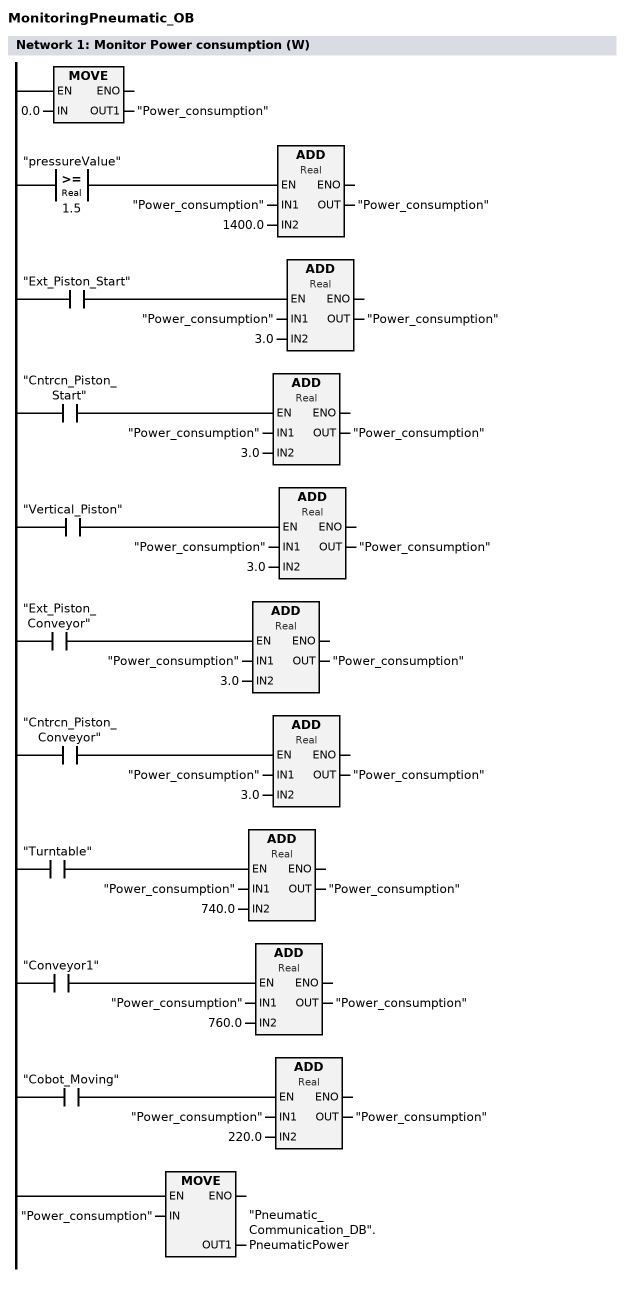
   RUNG wire#powerrail
      Move(in := 0.0, out1 => "Power_consumption")
   END_RUNG
   RUNG wire#powerrail
      { S7_Templates := "SrcType := Real" } GE_Contact(in1 := "pressureValue", in2 := 1.5)
      { S7_Templates := "SrcType := Real" } Add(in1 := "Power_consumption", in2 := 1400.0, out => "Power_consumption")
   END_RUNG
   RUNG wire#powerrail
      Contact( "Ext_Piston_Start" )
      { S7_Templates := "SrcType := Real" } Add(in1 := "Power_consumption", in2 := 3.0, out => "Power_consumption")
   END_RUNG
   RUNG wire#powerrail
      Contact( "Cntrcn_Piston_Start" )
      { S7_Templates := "SrcType := Real" } Add(in1 := "Power_consumption", in2 := 3.0, out => "Power_consumption")
   END_RUNG
   RUNG wire#powerrail
      Contact( "Vertical_Piston" )
      { S7_Templates := "SrcType := Real" } Add(in1 := "Power_consumption", in2 := 3.0, out => "Power_consumption")
   END_RUNG
   RUNG wire#powerrail
      Contact( "Ext_Piston_Conveyor" )
      { S7_Templates := "SrcType := Real" } Add(in1 := "Power_consumption", in2 := 3.0, out => "Power_consumption")
   END_RUNG
   RUNG wire#powerrail
      Contact( "Cntrcn_Piston_Conveyor" )
      { S7_Templates := "SrcType := Real" } Add(in1 := "Power_consumption", in2 := 3.0, out => "Power_consumption")
   END_RUNG
   RUNG wire#powerrail
      Contact( "Turntable" )
      { S7_Templates := "SrcType := Real" } Add(in1 := "Power_consumption", in2 := 740.0, out => "Power_consumption")
   END_RUNG
   RUNG wire#powerrail
      Contact( "Conveyor1" )
      { S7_Templates := "SrcType := Real" } Add(in1 := "Power_consumption", in2 := 760.0, out => "Power_consumption")
   END_RUNG
   RUNG wire#powerrail
      Contact( "Cobot_Moving" )
      { S7_Templates := "SrcType := Real" } Add(in1 := "Power_consumption", in2 := 220.0, out => "Power_consumption")
   END_RUNG
   RUNG wire#powerrail
      Move(in := "Power_consumption", out1 => "Pneumatic_Communication_DB".PneumaticPower)
   END_RUNG
   // the same network as SCL:
   "Power_consumption" := 0.0;
   IF "pressureValue" >= 1.5 THEN "Power_consumption" := "Power_consumption" + 1400.0; END_IF;
   IF "Ext_Piston_Start" THEN "Power_consumption" := "Power_consumption" + 3.0; END_IF;
   IF "Cntrcn_Piston_Start" THEN "Power_consumption" := "Power_consumption" + 3.0; END_IF;
   IF "Vertical_Piston" THEN "Power_consumption" := "Power_consumption" + 3.0; END_IF;
   IF "Ext_Piston_Conveyor" THEN "Power_consumption" := "Power_consumption" + 3.0; END_IF;
   IF "Cntrcn_Piston_Conveyor" THEN "Power_consumption" := "Power_consumption" + 3.0; END_IF;
   IF "Turntable" THEN "Power_consumption" := "Power_consumption" + 740.0; END_IF;
   IF "Conveyor1" THEN "Power_consumption" := "Power_consumption" + 760.0; END_IF;
   IF "Cobot_Moving" THEN "Power_consumption" := "Power_consumption" + 220.0; END_IF;
   "Pneumatic_Communication_DB".PneumaticPower := "Power_consumption";
END_REGION
END_ORGANIZATION_BLOCK

ORGANIZATION_BLOCK "RFID_OB"   // OB126, LAD, ProgramCycle
TITLE = "Main Program Sweep (Cycle)"
{ S7_Optimized_Access := 'TRUE' }
VERSION : 0.1
   VAR_INPUT
      Initial_Call : Bool;   // Initial call of this OB
      Remanence : Bool;   // =True, if remanent data are available
   END_VAR
   VAR_TEMP   // added for the SCL form of the ladder/FBD networks
      _w1 : Bool;
   END_VAR
BEGIN

REGION Network 1: Read nibble from RFID relay Device
   // K1 is LSB
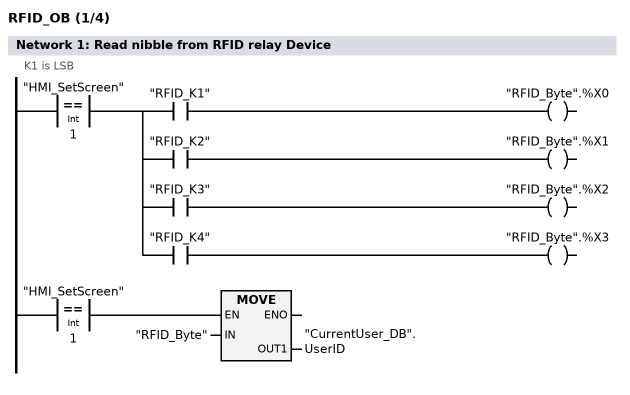
   RUNG wire#powerrail
      { S7_Templates := "SrcType := Int" } EQ_Contact(in1 := "HMI_SetScreen", in2 := 1)
      wire#w1
      Contact( "RFID_K1" )
      Coil( "RFID_Byte".%X0 )
   END_RUNG
   RUNG wire#w1
      Contact( "RFID_K2" )
      Coil( "RFID_Byte".%X1 )
   END_RUNG
   RUNG wire#w1
      Contact( "RFID_K3" )
      Coil( "RFID_Byte".%X2 )
   END_RUNG
   RUNG wire#w1
      Contact( "RFID_K4" )
      Coil( "RFID_Byte".%X3 )
   END_RUNG
   RUNG wire#powerrail
      { S7_Templates := "SrcType := Int" } EQ_Contact(in1 := "HMI_SetScreen", in2 := 1)
      Move(in := "RFID_Byte", out1 => "CurrentUser_DB".UserID)
   END_RUNG
   // the same network as SCL:
   #_w1 := "HMI_SetScreen" = 1;
   "RFID_Byte".%X0 := #_w1 AND "RFID_K1";
   "RFID_Byte".%X1 := #_w1 AND "RFID_K2";
   "RFID_Byte".%X2 := #_w1 AND "RFID_K3";
   "RFID_Byte".%X3 := #_w1 AND "RFID_K4";
   IF "HMI_SetScreen" = 1 THEN "CurrentUser_DB".UserID := "RFID_Byte"; END_IF;
END_REGION

REGION Network 2: Grant access and credentials
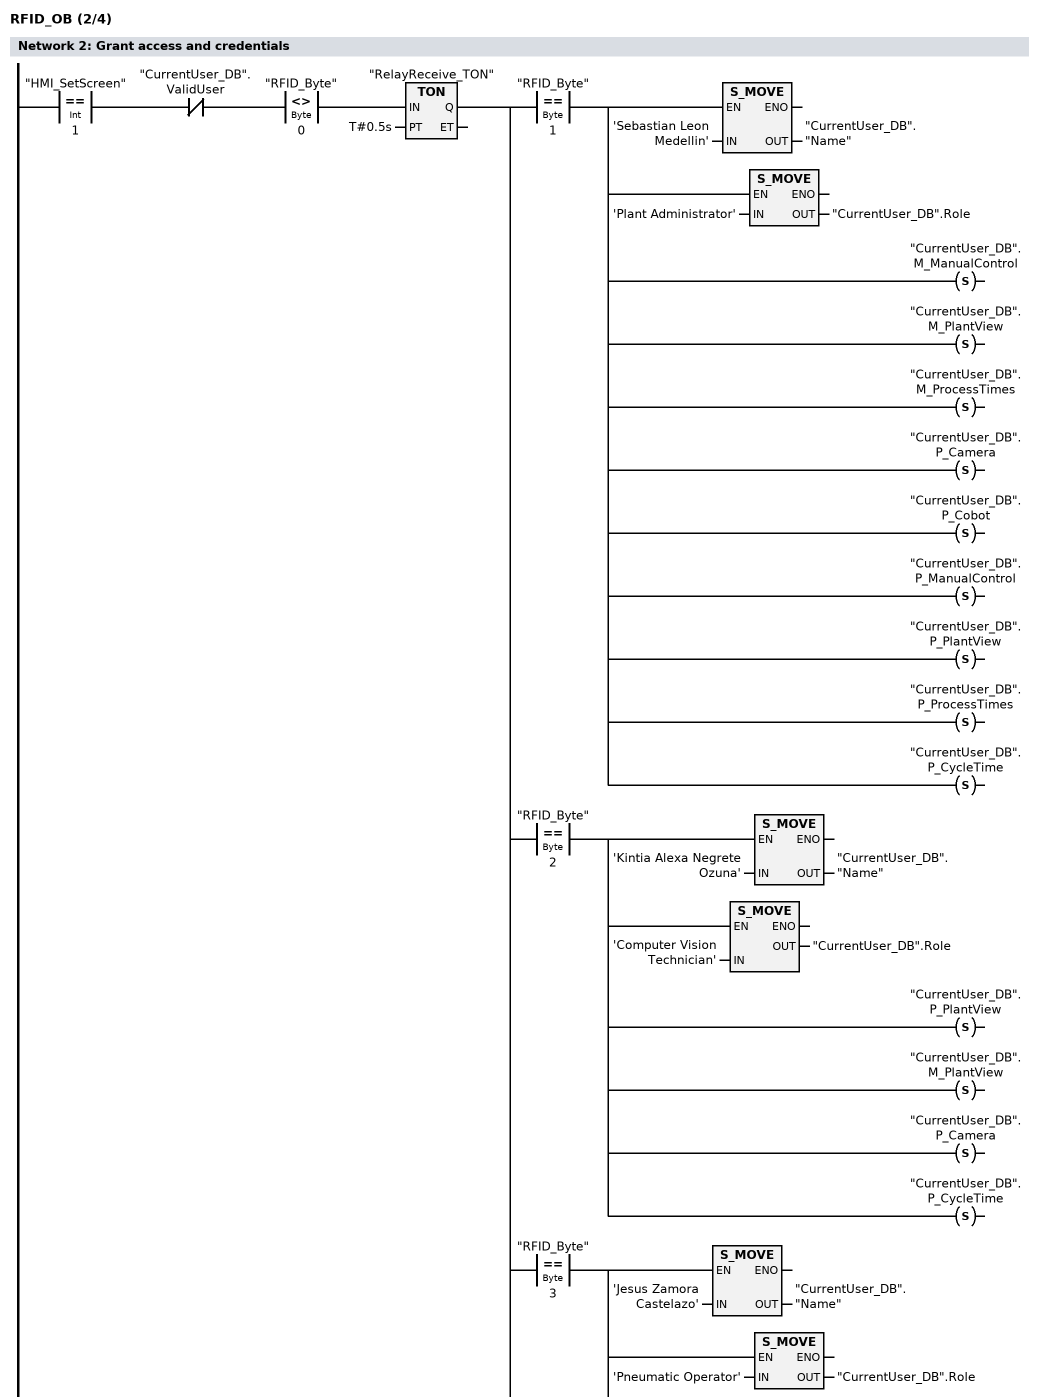
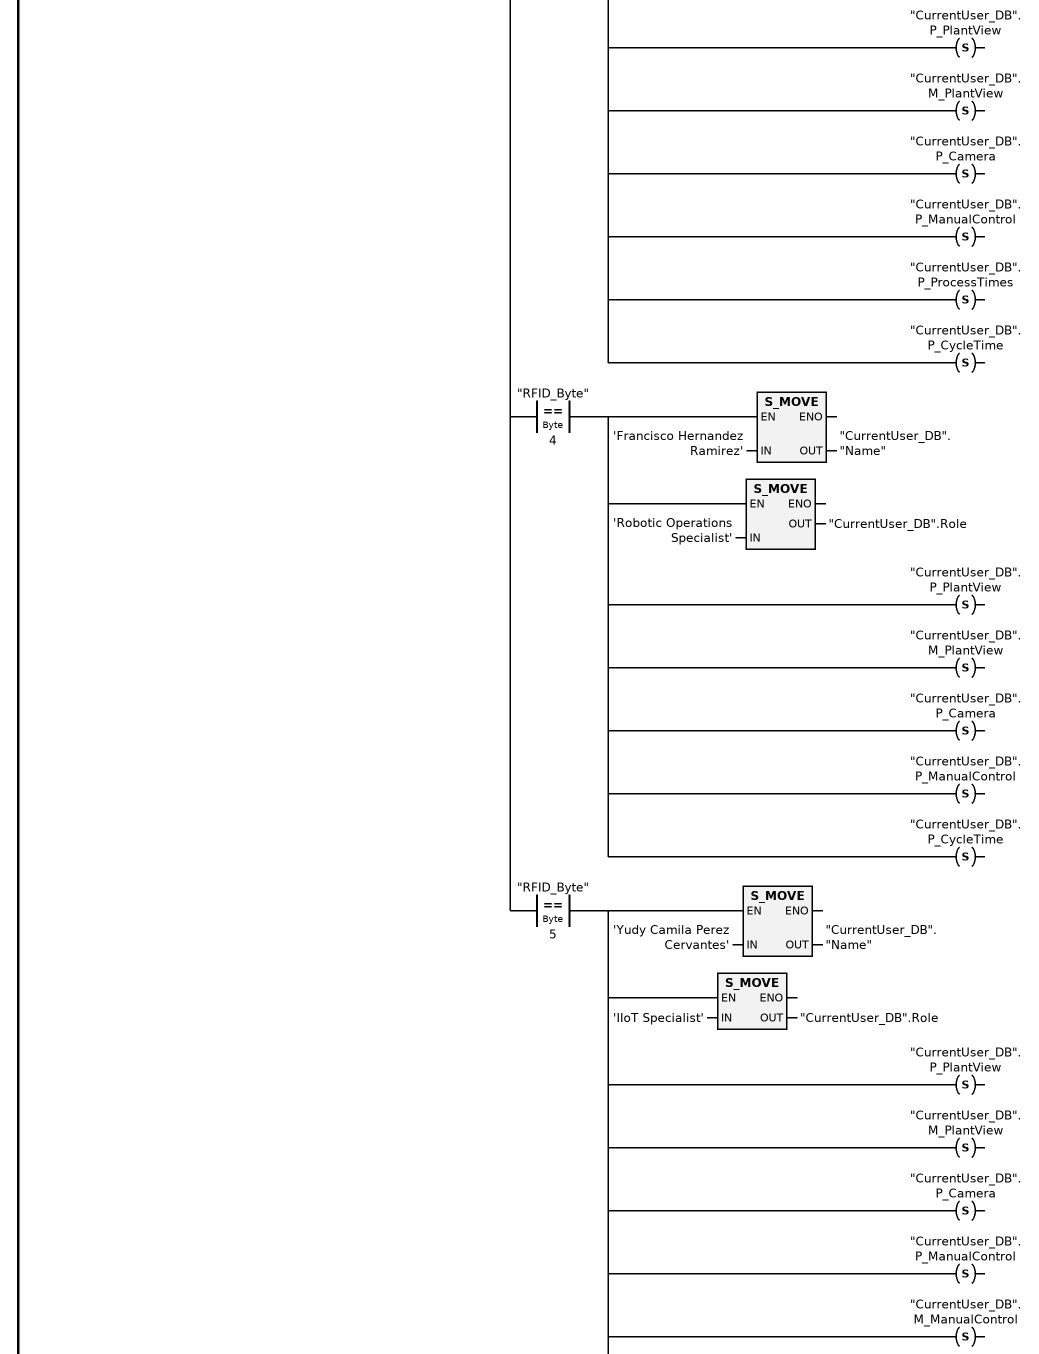
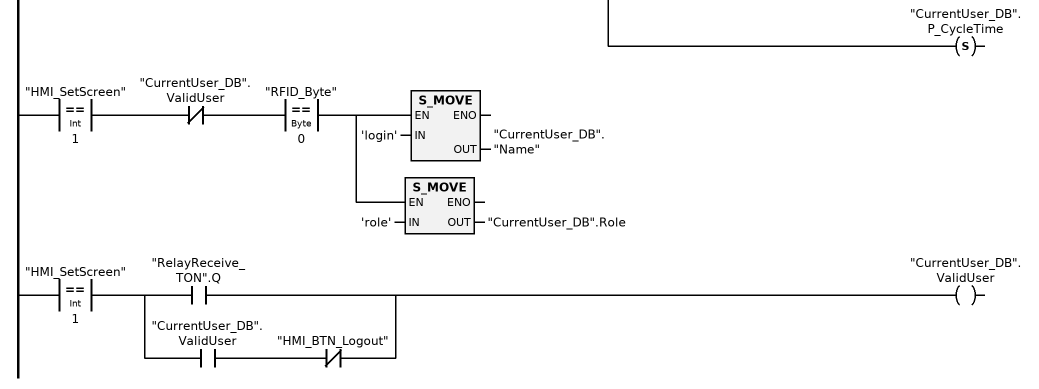
   "RelayReceive_TON".TON(IN := ("HMI_SetScreen" = 1) AND NOT "CurrentUser_DB".ValidUser AND ("RFID_Byte" <> 0),
                          PT := T#0.5s);
   IF "RelayReceive_TON".Q AND ("RFID_Byte" = 1) THEN
       "CurrentUser_DB"."Name" := 'Sebastian Leon Medellin';
       "CurrentUser_DB".Role := 'Plant Administrator';
       "CurrentUser_DB".M_ManualControl := TRUE;
       "CurrentUser_DB".M_PlantView := TRUE;
       "CurrentUser_DB".M_ProcessTimes := TRUE;
       "CurrentUser_DB".P_Camera := TRUE;
       "CurrentUser_DB".P_Cobot := TRUE;
       "CurrentUser_DB".P_ManualControl := TRUE;
       "CurrentUser_DB".P_PlantView := TRUE;
       "CurrentUser_DB".P_ProcessTimes := TRUE;
       "CurrentUser_DB".P_CycleTime := TRUE;
   END_IF;
   IF "RelayReceive_TON".Q AND ("RFID_Byte" = 2) THEN
       "CurrentUser_DB"."Name" := 'Kintia Alexa Negrete Ozuna';
       "CurrentUser_DB".Role := 'Computer Vision Technician';
       "CurrentUser_DB".P_PlantView := TRUE;
       "CurrentUser_DB".M_PlantView := TRUE;
       "CurrentUser_DB".P_Camera := TRUE;
       "CurrentUser_DB".P_CycleTime := TRUE;
   END_IF;
   IF "RelayReceive_TON".Q AND ("RFID_Byte" = 3) THEN
       "CurrentUser_DB"."Name" := 'Jesus Zamora Castelazo';
       "CurrentUser_DB".Role := 'Pneumatic Operator';
       "CurrentUser_DB".P_PlantView := TRUE;
       "CurrentUser_DB".M_PlantView := TRUE;
       "CurrentUser_DB".P_Camera := TRUE;
       "CurrentUser_DB".P_ManualControl := TRUE;
       "CurrentUser_DB".P_ProcessTimes := TRUE;
       "CurrentUser_DB".P_CycleTime := TRUE;
   END_IF;
   IF "RelayReceive_TON".Q AND ("RFID_Byte" = 4) THEN
       "CurrentUser_DB"."Name" := 'Francisco Hernandez Ramirez';
       "CurrentUser_DB".Role := 'Robotic Operations Specialist';
       "CurrentUser_DB".P_PlantView := TRUE;
       "CurrentUser_DB".M_PlantView := TRUE;
       "CurrentUser_DB".P_Camera := TRUE;
       "CurrentUser_DB".P_ManualControl := TRUE;
       "CurrentUser_DB".P_CycleTime := TRUE;
   END_IF;
   IF "RelayReceive_TON".Q AND ("RFID_Byte" = 5) THEN
       "CurrentUser_DB"."Name" := 'Yudy Camila Perez Cervantes';
       "CurrentUser_DB".Role := 'IIoT Specialist';
       "CurrentUser_DB".P_PlantView := TRUE;
       "CurrentUser_DB".M_PlantView := TRUE;
       "CurrentUser_DB".P_Camera := TRUE;
       "CurrentUser_DB".P_ManualControl := TRUE;
       "CurrentUser_DB".M_ManualControl := TRUE;
       "CurrentUser_DB".P_CycleTime := TRUE;
   END_IF;
   IF ("HMI_SetScreen" = 1) AND NOT "CurrentUser_DB".ValidUser AND ("RFID_Byte" = 0) THEN
       "CurrentUser_DB"."Name" := 'login';
       "CurrentUser_DB".Role := 'role';
   END_IF;
   "CurrentUser_DB".ValidUser := ("HMI_SetScreen" = 1) AND ("RelayReceive_TON".Q OR ("CurrentUser_DB".ValidUser AND NOT "HMI_BTN_Logout"));
END_REGION

REGION Network 3: Send user and role data trough S7
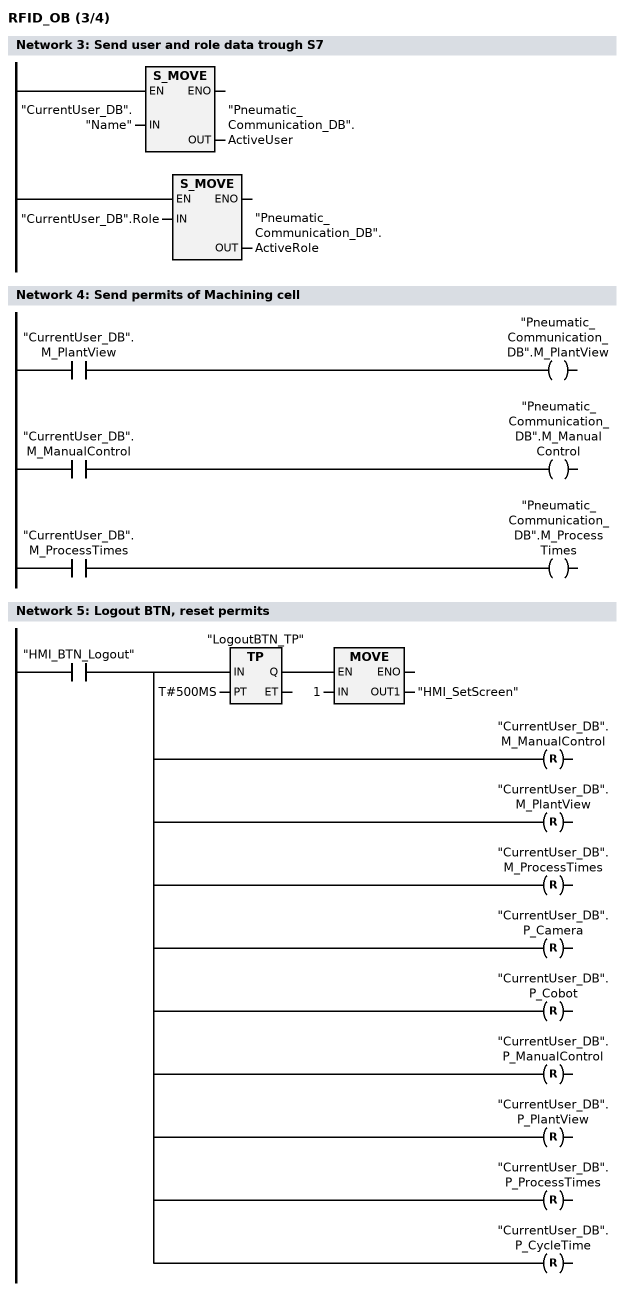
   RUNG wire#powerrail
      S_Move(in := "CurrentUser_DB"."Name", out => "Pneumatic_Communication_DB".ActiveUser)
   END_RUNG
   RUNG wire#powerrail
      S_Move(in := "CurrentUser_DB".Role, out => "Pneumatic_Communication_DB".ActiveRole)
   END_RUNG
   // the same network as SCL:
   "Pneumatic_Communication_DB".ActiveUser := "CurrentUser_DB"."Name";
   "Pneumatic_Communication_DB".ActiveRole := "CurrentUser_DB".Role;
END_REGION

REGION Network 4: Send permits of Machining cell
   RUNG wire#powerrail
      Contact( "CurrentUser_DB".M_PlantView )
      Coil( "Pneumatic_Communication_DB".M_PlantView )
   END_RUNG
   RUNG wire#powerrail
      Contact( "CurrentUser_DB".M_ManualControl )
      Coil( "Pneumatic_Communication_DB".M_ManualControl )
   END_RUNG
   RUNG wire#powerrail
      Contact( "CurrentUser_DB".M_ProcessTimes )
      Coil( "Pneumatic_Communication_DB".M_ProcessTimes )
   END_RUNG
   // the same network as SCL:
   "Pneumatic_Communication_DB".M_PlantView := "CurrentUser_DB".M_PlantView;
   "Pneumatic_Communication_DB".M_ManualControl := "CurrentUser_DB".M_ManualControl;
   "Pneumatic_Communication_DB".M_ProcessTimes := "CurrentUser_DB".M_ProcessTimes;
END_REGION

REGION Network 5: Logout BTN, reset permits
   "LogoutBTN_TP".TP(IN := "HMI_BTN_Logout", PT := T#500MS);
   IF "LogoutBTN_TP".Q THEN "HMI_SetScreen" := 1; END_IF;
   IF "HMI_BTN_Logout" THEN
       "CurrentUser_DB".M_ManualControl := FALSE;
       "CurrentUser_DB".M_PlantView := FALSE;
       "CurrentUser_DB".M_ProcessTimes := FALSE;
       "CurrentUser_DB".P_Camera := FALSE;
       "CurrentUser_DB".P_Cobot := FALSE;
       "CurrentUser_DB".P_ManualControl := FALSE;
       "CurrentUser_DB".P_PlantView := FALSE;
       "CurrentUser_DB".P_ProcessTimes := FALSE;
       "CurrentUser_DB".P_CycleTime := FALSE;
   END_IF;
END_REGION

REGION Network 6: Send logout bit
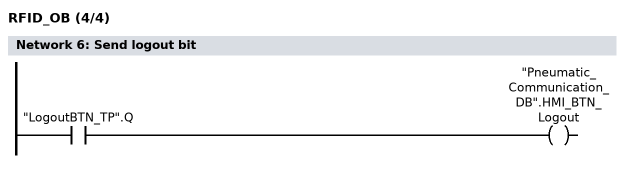
   RUNG wire#powerrail
      Contact( "LogoutBTN_TP".Q )
      Coil( "Pneumatic_Communication_DB".HMI_BTN_Logout )
   END_RUNG
   // the same network as SCL:
   "Pneumatic_Communication_DB".HMI_BTN_Logout := "LogoutBTN_TP".Q;
END_REGION
END_ORGANIZATION_BLOCK

ORGANIZATION_BLOCK "CycleTime_OB"   // OB127, LAD, ProgramCycle
TITLE = "Main Program Sweep (Cycle)"
{ S7_Optimized_Access := 'TRUE' }
VERSION : 0.1
   VAR_INPUT
      Initial_Call : Bool;   // Initial call of this OB
      Remanence : Bool;   // =True, if remanent data are available
   END_VAR
BEGIN

REGION Network 1: Enabled Measuring latch
   // This latch confirms that the PLC is either
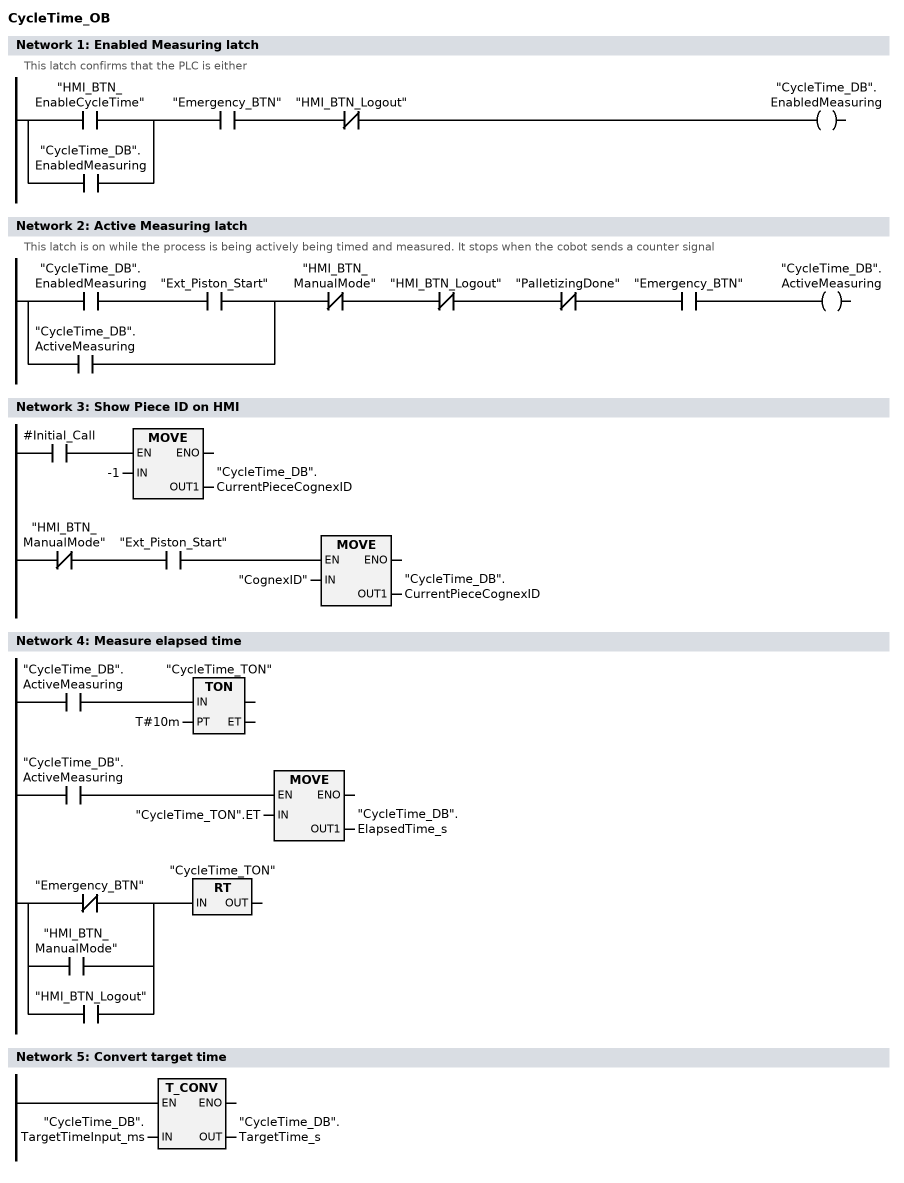
   RUNG wire#powerrail
      Contact( "HMI_BTN_EnableCycleTime" )
      wire#w1
      Contact( "Emergency_BTN" )
      I_Contact( "HMI_BTN_Logout" )
      Coil( "CycleTime_DB".EnabledMeasuring )
   END_RUNG
   RUNG wire#powerrail
      Contact( "CycleTime_DB".EnabledMeasuring )
   END_RUNG wire#w1
   // the same network as SCL:
   "CycleTime_DB".EnabledMeasuring := ("HMI_BTN_EnableCycleTime" OR "CycleTime_DB".EnabledMeasuring) AND "Emergency_BTN" AND NOT "HMI_BTN_Logout";
END_REGION

REGION Network 2: Active Measuring latch
   // This latch is on while the process is being actively being timed and measured. It stops when the cobot sends a counter signal
   RUNG wire#powerrail
      Contact( "CycleTime_DB".EnabledMeasuring )
      Contact( "Ext_Piston_Start" )
      wire#w1
      I_Contact( "HMI_BTN_ManualMode" )
      I_Contact( "HMI_BTN_Logout" )
      I_Contact( "PalletizingDone" )
      Contact( "Emergency_BTN" )
      Coil( "CycleTime_DB".ActiveMeasuring )
   END_RUNG
   RUNG wire#powerrail
      Contact( "CycleTime_DB".ActiveMeasuring )
   END_RUNG wire#w1
   // the same network as SCL:
   "CycleTime_DB".ActiveMeasuring := (("CycleTime_DB".EnabledMeasuring AND "Ext_Piston_Start") OR "CycleTime_DB".ActiveMeasuring) AND NOT "HMI_BTN_ManualMode" AND NOT "HMI_BTN_Logout" AND NOT "PalletizingDone" AND "Emergency_BTN";
END_REGION

REGION Network 3: Show Piece ID on HMI
   RUNG wire#powerrail
      Contact( #Initial_Call )
      Move(in := -1, out1 => "CycleTime_DB".CurrentPieceCognexID)
   END_RUNG
   RUNG wire#powerrail
      I_Contact( "HMI_BTN_ManualMode" )
      Contact( "Ext_Piston_Start" )
      Move(in := "CognexID", out1 => "CycleTime_DB".CurrentPieceCognexID)
   END_RUNG
   // the same network as SCL:
   IF #Initial_Call THEN "CycleTime_DB".CurrentPieceCognexID := -1; END_IF;
   IF NOT "HMI_BTN_ManualMode" AND "Ext_Piston_Start" THEN
       "CycleTime_DB".CurrentPieceCognexID := "CognexID";
   END_IF;
END_REGION

REGION Network 4: Measure elapsed time
   "CycleTime_TON".TON(IN := "CycleTime_DB".ActiveMeasuring, PT := T#10m);
   IF "CycleTime_DB".ActiveMeasuring THEN "CycleTime_DB".ElapsedTime_s := "CycleTime_TON".ET; END_IF;
   IF NOT "Emergency_BTN" OR "HMI_BTN_ManualMode" OR "HMI_BTN_Logout" THEN
       RESET_TIMER("CycleTime_TON");
   END_IF;
END_REGION

REGION Network 5: Convert target time
   "CycleTime_DB".TargetTime_s := T_CONV(IN := "CycleTime_DB".TargetTimeInput_ms);
END_REGION
END_ORGANIZATION_BLOCK

(* ===== HMI "HMI_RT_1" =====
system functions are stored by id; their names below are inferred from use
connection "HMI_Connection_1": ETHERNET, SMART_S7_1200_OMS

HMI tags "Default tag table"
   "Tag_ScreenNumber" : UInt, internal
   "HMI_BTN1" : Bool = PLC HMI_BTN1 AT %M50.0, 100 ms
   "Conveyor2" : Bool = PLC Conveyor2 AT %Q0.0, 100 ms
   "Pusher1" : Bool = PLC Pusher1 AT %Q0.1, 100 ms
   "Drill" : Bool = PLC Drill AT %Q0.3, 100 ms
   "Mix" : Bool = PLC Mix AT %Q0.5, 100 ms
   "Pusher2" : Bool = PLC Pusher2 AT %Q0.6, 500 ms
   "Conveyor5" : Bool = PLC Conveyor5 AT %Q0.7, 100 ms
   "Conveyor6_OUT" : Bool = PLC Conveyor6_OUT AT %Q8.3, 100 ms
   "Conveyor6_IN" : Bool = PLC Conveyor6_IN AT %Q8.2, 100 ms
   "Red_Tower" : Bool = PLC Red_Tower AT %Q1.1, 500 ms
   "Green_Tower" : Bool = PLC Green_Tower AT %Q1.0, 100 ms
   "cakeFlavor" : UInt = PLC cakeFlavor AT %MW12, 100 ms
   "Conveyor3" : Bool = PLC Conveyor3 AT %Q0.2, 100 ms
   "Conveyor4" : Bool = PLC Conveyor4 AT %Q0.4, 100 ms
   "Press_UP" : Bool = PLC Press_UP AT %Q8.4, 100 ms
   "Press_DOWN" : Bool = PLC Press_DOWN AT %Q8.5, 100 ms
   "drillingTime" : Time = PLC drillingTime AT %MD14, 100 ms
   "processTimes_DB_chocolateDrillingInput" : UInt = PLC processTimes_DB.chocolateDrillingInput_ms, 1 s
   "processTimes_DB_chocolateMixingInput" : UInt = PLC processTimes_DB.chocolateMixingInput_ms, 1 s
   "processTimes_DB_vanillaDrillingInput_ms" : UInt = PLC processTimes_DB.vanillaDrillingInput_ms, 1 s
   "processTimes_DB_vamillaMixingInput_ms" : UInt = PLC processTimes_DB.vanillaMixingInput_ms, 1 s
   "processTimes_DB_strawberryDrillingInput_ms" : UInt = PLC processTimes_DB.strawberryDrillingInput_ms, 1 s
   "processTimes_DB_strawberryMixingInput_ms" : UInt = PLC processTimes_DB.strawberryMixingInput_ms, 1 s
   "ManualMode_SW" : Bool = PLC ManualMode_SW AT %M53.0, 100 ms
   "HMI_BTN_Conveyor2" : Bool = PLC HMI_BTN_Conveyor2 AT %M50.1, 100 ms
   "HMI_BTN_Pusher1" : Bool = PLC HMI_BTN_Pusher1 AT %M50.2, 100 ms
   "HMI_BTN_Conveyor3" : Bool = PLC HMI_BTN_Conveyor3 AT %M50.3, 100 ms
   "HMI_BTN_Conveyor4" : Bool = PLC HMI_BTN_Conveyor4 AT %M50.4, 100 ms
   "HMI_BTN_Drill" : Bool = PLC HMI_BTN_Drill AT %M50.6, 100 ms
   "HMI_BTN_Mix" : Bool = PLC HMI_BTN_Mix AT %M50.7, 100 ms
   "HMI_BTN_Conveyor5" : Bool = PLC HMI_BTN_Conveyor5 AT %M50.5, 100 ms
   "HMI_BTN_Pusher2" : Bool = PLC HMI_BTN_Pusher2 AT %M51.0, 100 ms
   "HMI_BTN_Conveyor6IN" : Bool = PLC HMI_BTN_Conveyor6IN AT %M51.1, 100 ms
   "HMI_BTN_Conveyor6OUT" : Bool = PLC HMI_BTN_Conveyor6OUT AT %M51.2, 100 ms
   "HMI_BTN_PressDown" : Bool = PLC HMI_BTN_PressDown AT %M51.3, 100 ms
   "HMI_BTN_PressUp" : Bool = PLC HMI_BTN_PressUp AT %M51.4, 100 ms
   "Power_consumption" : Real = PLC Power_consumption AT %MD28, 100 ms
   "HMI_SetScreen" : Int = PLC HMI_SetScreen AT %MW54, 100 ms
      on ChangeValue: ActivateScreenByNumber("HMI_SetScreen", 0)
   "HMI_BTN_PlantView" : Bool = PLC HMI_BTN_PlantView AT %M51.5, 100 ms
   "HMI_BTN_ProcessTimes" : Bool = PLC HMI_BTN_ProcessTimes AT %M51.6, 100 ms
   "HMI_BTN_ManualControl" : Bool = PLC HMI_BTN_ManualControl AT %M51.7, 100 ms
   "Machining_Communication_DB_M_PlantView" : Bool = PLC Machining_Communication_DB.M_PlantView AT %DB100.DBX5.5, 1 s
   "Machining_Communication_DB_M_ProcessTimes" : Bool = PLC Machining_Communication_DB.M_ProcessTimes AT %DB100.DBX5.7, 1 s
   "Machining_Communication_DB_M_ManualControl" : Bool = PLC Machining_Communication_DB.M_ManualControl AT %DB100.DBX5.6, 1 s

text list "Flavors": 0 'Chocolate'; 1 'Vanilla'; 2 'Strawberry'; 4 'Flavor'; -1 'NA'

Template "Template_1" 800x480
   TextField "Template_Text field_1" at 62,8 size 412x56; Text 'MR2007B Automation of Manufacturing Systems ATOLE S.A. de C.V.'
   GraphicView "Template_Graphic view_1" at 529,9 size 252x54; Picture "eic"
   GraphicView "Template_Graphic view_2" at 21,13 size 34x45; Picture "atoleLogo_transparent"

screen "Root screen" 800x480, template "Template_1"
   TextField "HmiScreenItemData" at 40,88 size 720x57; Text 'Welcome to ATOLE S.A. de C.V.'
   Button "Button_2" at 136,208 size 240x56; TextOff 'Plant View'
      on Press: SetBit("HMI_BTN_PlantView")
      on Release: ResetBit("HMI_BTN_PlantView")
   GraphicView "Graphic view_1" at 429,152 size 294x294; Picture "cake"
   Button "Button_3" at 136,280 size 240x56; TextOff 'Set Process Times'
      on Press: SetBit("HMI_BTN_ProcessTimes")
      on Release: ResetBit("HMI_BTN_ProcessTimes")
   Button "Button_4" at 136,352 size 240x56; TextOff 'Manual Control'
      on Press: SetBit("HMI_BTN_ManualControl")
      on Release: ResetBit("HMI_BTN_ManualControl")
   Rectangle "Rectangle_1" at 144,216 size 40x40
      Appearance <- "Machining_Communication_DB_M_PlantView"
   Rectangle "Rectangle_2" at 144,288 size 40x40
      Appearance <- "Machining_Communication_DB_M_ProcessTimes"
   Rectangle "Rectangle_3" at 144,360 size 40x40
      Appearance <- "Machining_Communication_DB_M_ManualControl"

screen "PlantView" 800x480, template "Template_1"
   GraphicView "Graphic view_1" at 14,74 size 773x401; Picture "machiningCellDiagram_2"
   Circle "Circle_1" at 684,86 size 11x11
      Visibility <- "Conveyor2"
   Circle "Circle_2" at 747,252 size 11x11
      Visibility <- "Pusher1"
   Circle "Circle_3" at 546,386 size 11x11
      Visibility <- "Drill"
   Circle "Circle_4" at 323,435 size 11x11
      Visibility <- "Pusher2"
   Circle "Circle_5" at 342,144 size 11x11
      Visibility <- "Conveyor5"
   Circle "Circle_6" at 400,386 size 11x11
      Visibility <- "Mix"
   GraphicView "Graphic view_2" at 33,112 size 21x24; Picture "arrow"
      Visibility <- "Conveyor6_OUT"
   GraphicView "Graphic view_3" at 33,186 size 21x24; Picture "arrowDown"
      Visibility <- "Conveyor6_IN"
   Rectangle "Rectangle_1" at 670,360 size 20x20
      Visibility <- "Red_Tower"
   Rectangle "Rectangle_2" at 699,360 size 20x20
      Visibility <- "Green_Tower"
   TextField "Text field_1" at 319,72 size 162x39; Text 'Plant View'
   Circle "Circle_7" at 556,194 size 11x11
      Visibility <- "Conveyor3"
   Circle "Circle_8" at 417,194 size 11x11
      Visibility <- "Conveyor4"
   GraphicView "Graphic view_4" at 33,361 size 21x24; Picture "arrowDown"
      Visibility <- "Press_DOWN"
   GraphicView "Graphic view_5" at 33,286 size 21x24; Picture "arrow"
      Visibility <- "Press_UP"
   IOField "I/O field_1" at 600,432 size 184x32; FormatPattern 999999999999; Unit  W
      ProcessValue <- "Power_consumption"
   TextField "Text field_2" at 616,408 size 168x23; Text 'Power Consumption'
   Button "Button_1" at 16,424 size 104x40; TextOff 'Home'
      on Press: ActivateScreen("Root screen", 0); SetTag("HMI_SetScreen", 2)

screen "ManualControl" 800x480, template "Template_1"
   Switch "Switch_1" at 84,224 size 120x56; CaptionText 'Switch'; TextOff 'OFF'; TextOn 'ON'
      ProcessValue <- "ManualMode_SW"
      on SwitchOn: SetBit("ManualMode_SW")
      on SwitchOff: ResetBit("ManualMode_SW")
   TextField "Text field_2" at 84,284 size 121x36; Text 'Enable manual control'
   Button "Button_2" at 252,144 size 144x32; TextOff 'Conveyor 2'
      on Press: SetBit("HMI_BTN_Conveyor2")
      on Release: ResetBit("HMI_BTN_Conveyor2")
   Button "Button_3" at 252,192 size 144x32; TextOff 'Pusher 1'
      on Press: SetBit("HMI_BTN_Pusher1")
      on Release: ResetBit("HMI_BTN_Pusher1")
   Button "Button_4" at 252,240 size 144x32; TextOff 'Conveyor 3'
      on Release: ResetBit("HMI_BTN_Conveyor3")
      on Press: SetBit("HMI_BTN_Conveyor3")
   Button "Button_5" at 252,288 size 144x32; TextOff 'Conveyor 4'
      on Press: SetBit("HMI_BTN_Conveyor4")
      on Release: ResetBit("HMI_BTN_Conveyor4")
   Button "Button_6" at 252,336 size 144x32; TextOff 'Drill'
      on Press: SetBit("HMI_BTN_Drill")
      on Release: ResetBit("HMI_BTN_Drill")
   Button "Button_7" at 252,384 size 144x32; TextOff 'Mix'
      on Press: SetBit("HMI_BTN_Mix")
      on Release: ResetBit("HMI_BTN_Mix")
   Button "Button_8" at 524,144 size 144x32; TextOff 'Pusher 2'
      on Press: SetBit("HMI_BTN_Pusher2")
      on Release: ResetBit("HMI_BTN_Pusher2")
   Button "Button_9" at 524,192 size 144x32; TextOff 'Conveyor 5'
      on Press: SetBit("HMI_BTN_Conveyor5")
      on Release: ResetBit("HMI_BTN_Conveyor5")
   Circle "Circle_1" at 412,144 size 32x32
      Appearance <- "Conveyor2"
   Circle "Circle_2" at 412,192 size 32x32
      Appearance <- "Pusher1"
   Circle "Circle_3" at 412,240 size 32x32
      Appearance <- "Conveyor3"
   Circle "Circle_4" at 412,288 size 32x32
      Appearance <- "Conveyor4"
   Circle "Circle_5" at 412,336 size 32x32
      Appearance <- "Drill"
   Circle "Circle_6" at 412,384 size 32x32
      Appearance <- "Mix"
   Circle "Circle_7" at 684,144 size 32x32
      Appearance <- "Pusher2"
   Circle "Circle_8" at 684,192 size 32x32
      Appearance <- "Conveyor5"
   Button "Button_10" at 524,240 size 144x32; TextOff 'Conveyor 6 IN'
      on Press: SetBit("HMI_BTN_Conveyor6IN")
      on Release: ResetBit("HMI_BTN_Conveyor6IN")
   Button "Button_11" at 524,288 size 144x32; TextOff 'Conveyor 6 OUT'
      on Press: SetBit("HMI_BTN_Conveyor6OUT")
      on Release: ResetBit("HMI_BTN_Conveyor6OUT")
   Button "Button_12" at 524,336 size 144x32; TextOff 'Press Down'
      on Press: SetBit("HMI_BTN_PressDown")
      on Release: ResetBit("HMI_BTN_PressDown")
   Button "Button_13" at 524,384 size 144x32; TextOff 'Press Up'
      on Press: SetBit("HMI_BTN_PressUp")
      on Release: ResetBit("HMI_BTN_PressUp")
   Circle "Circle_9" at 684,240 size 32x32
      Appearance <- "Conveyor6_IN"
   Circle "Circle_10" at 684,288 size 32x32
      Appearance <- "Conveyor6_OUT"
   Circle "Circle_11" at 684,336 size 32x32
      Appearance <- "Press_DOWN"
   Circle "Circle_12" at 684,384 size 32x32
      Appearance <- "Press_UP"
   Button "Button_1" at 16,424 size 104x40; TextOff 'Home'
      on Press: ActivateScreen("Root screen", 0); SetTag("HMI_SetScreen", 2)
   TextField "Text field_1" at 208,80 size 389x39; Text 'Machining Manual Control'
   Group "Group" at 84,144 size 632x272
   TextField "Text field_4" at 400,432 size 393x48; Text 'Manual Mode: Press and hold the button to actuate'

screen "ProcessTimes" 800x480, template "Template_1"
   TextField "Text field_1" at 294,88 size 213x39; Text 'Process Times'
   Button "Button_1" at 16,424 size 104x40; TextOff 'Home'
      on Press: ActivateScreen("Root screen", 0); SetTag("HMI_SetScreen", 2)
   TextField "Text field_5" at 74,208 size 104x48; Text 'Drilling'
   TextField "Text field_6" at 82,280 size 96x48; Text 'Mixing'
   IOField "I/O field_1" at 190,208 size 152x48; FormatPattern 9999999; Unit  s
      ProcessValue <- "processTimes_DB_chocolateDrillingInput"
   IOField "I/O field_2" at 190,280 size 152x48; FormatPattern 9999999; Unit  s
      ProcessValue <- "processTimes_DB_chocolateMixingInput"
   TextField "Text field_2" at 190,168 size 156x34; Text 'Chocolate'
   TextField "Text field_3" at 382,168 size 156x34; Text 'Vanilla'
   TextField "Text field_4" at 574,168 size 152x31; Text 'Strawberry'
   IOField "I/O field_3" at 382,280 size 152x48; FormatPattern 9999999; Unit  s
      ProcessValue <- "processTimes_DB_vamillaMixingInput_ms"
   IOField "I/O field_4" at 382,208 size 152x48; FormatPattern 9999999; Unit  s
      ProcessValue <- "processTimes_DB_vanillaDrillingInput_ms"
   IOField "I/O field_5" at 574,208 size 152x48; FormatPattern 9999999; Unit  s
      ProcessValue <- "processTimes_DB_strawberryDrillingInput_ms"
   IOField "I/O field_6" at 574,280 size 152x48; FormatPattern 9999999; Unit  s
      ProcessValue <- "processTimes_DB_strawberryMixingInput_ms"

screen "Access_Screen" 800x480
   TextField "Text field_2" at 255,160 size 290x95; Text 'Please present your RFID card to the reader interface'
   GraphicView "Graphic view_1" at 320,224 size 160x152; Picture "rfidSym"
   TextField "Text field_1" at 262,40 size 276x47; Text 'Access Control'
*)

(* ===== HMI "HMI_RT_2" =====
system functions are stored by id; their names below are inferred from use
connection "HMI_Connection_2": ETHERNET, SMART_S7_1200_OMS

HMI tags "Default tag table"
   "Tag_ScreenNumber" : UInt, internal
   "Vertical_Piston" : Bool = PLC Vertical_Piston AT %Q8.5, 500 ms
   "ScanBTN_HMI" : Bool = PLC HMI_BTN_Scan AT %M51.2, 100 ms
   "Conveyor1" : Bool = PLC Conveyor1 AT %Q9.1, 100 ms
   "Cntrcn_Piston_Start" : Bool = PLC Cntrcn_Piston_Start AT %Q8.3, 100 ms
   "Ext_Piston_Start" : Bool = PLC Ext_Piston_Start AT %Q8.4, 100 ms
   "Turntable" : Bool = PLC Turntable AT %Q9.0, 500 ms
   "Ext_Piston_Conveyor" : Bool = PLC Ext_Piston_Conveyor AT %Q8.7, 100 ms
   "Cntrcn_Piston_Conveyor" : Bool = PLC Cntrcn_Piston_Conveyor AT %Q8.6, 100 ms
   "pressureValue" : Real = PLC pressureValue AT %MD34, 100 ms
   "HMI_BTN_Ext_Piston_Start" : Bool = PLC HMI_BTN_Ext_Piston_Start AT %M50.6, 100 ms
   "HMI_BTN_Cntrcn_Piston_Start" : Bool = PLC HMI_BTN_Cntrcn_Piston_Start AT %M50.5, 100 ms
   "HMI_BTN_Vertical_Piston" : Bool = PLC HMI_BTN_Vertical_Piston AT %M50.4, 100 ms
   "HMI_BTN_Turntable" : Bool = PLC HMI_BTN_Turntable AT %M51.1, 100 ms
   "HMI_BTN_Ext_Piston_Conveyor" : Bool = PLC HMI_BTN_Ext_Piston_Conveyor AT %M50.7, 100 ms
   "HMI_BTN_Cntrcn_Piston_Conveyor" : Bool = PLC HMI_BTN_Cntrcn_Piston_Conveyor AT %M50.3, 100 ms
   "HMI_BTN_Conveyor1" : Bool = PLC HMI_BTN_Conveyor1 AT %M51.0, 100 ms
   "HMI_BTN_ManualMode" : Bool = PLC HMI_BTN_ManualMode AT %M51.3, 100 ms
   "CognexId" : UInt = PLC CognexId_UInt AT %MW10, 100 ms
   "secondsSincePhoto" : DInt = PLC secondsSincePhoto AT %MD14, 100 ms
   "Pneumatic_Times_DB_chocolatePunchingInput_ms" : UInt = PLC Pneumatic_Times_DB.chocolatePunchingInput_ms, 1 s
   "Pneumatic_Times_DB_vanillaPunchingInput_ms" : UInt = PLC Pneumatic_Times_DB.vanillaPunchingInput_ms, 1 s
   "Pneumatic_Times_DB_strawberryPunchingInput_ms" : UInt = PLC Pneumatic_Times_DB.strawberryPunchingInput_ms, 1 s
   "Power_consumption" : Real = PLC Power_consumption AT %MD44, 100 ms
   "HMI_ShowBusyMessage" : Bool = PLC HMI_ShowBusyMessage AT %M51.4, 100 ms
   "CognexID(1)" : Int = PLC CognexID AT %MW20, 100 ms
   "HMI_CurrentScreen" : UInt = PLC HMI_CurrentScreen AT %MW52, 100 ms
   "HMI_SetScreen" : Int = PLC HMI_SetScreen AT %MW54, 100 ms
      on ChangeValue: ActivateScreenByNumber("HMI_SetScreen", 0)
   "HMI_BTN_Enter" : Bool = PLC HMI_BTN_Enter AT %M51.5, 100 ms
   "HMI_BTN_PlantView" : Bool = PLC HMI_BTN_PlantView AT %M51.6, 100 ms
   "HMI_BTN_ProcessTimes" : Bool = PLC HMI_BTN_ProcessTimes AT %M51.7, 100 ms
   "HMI_BTN_ManualModeScr" : Bool = PLC HMI_BTN_ManualModeScr AT %M56.0, 100 ms
   "HMI_BTN_CameraControl" : Bool = PLC HMI_BTN_CameraControl AT %M56.1, 100 ms
   "CurrentUser_DB_Name" : String[40] = PLC CurrentUser_DB.Name AT %DB11.DBX2.0, 100 ms
   "CurrentUser_DB_ValidUser" : Bool = PLC CurrentUser_DB.ValidUser AT %DB11.DBX71.0, 100 ms
   "HMI_BTN_Logout" : Bool = PLC HMI_BTN_Logout AT %M56.2, 100 ms
   "CurrentUser_DB_Role" : String[25] = PLC CurrentUser_DB.Role AT %DB11.DBX44.0, 100 ms
   "CurrentUser_DB_P_PlantView" : Bool = PLC CurrentUser_DB.P_PlantView AT %DB11.DBX71.1, 100 ms
   "CurrentUser_DB_P_ProcessTimes" : Bool = PLC CurrentUser_DB.P_ProcessTimes AT %DB11.DBX71.5, 100 ms
   "CurrentUser_DB_P_ManualControl" : Bool = PLC CurrentUser_DB.P_ManualControl AT %DB11.DBX71.2, 100 ms
   "CurrentUser_DB_P_Camera" : Bool = PLC CurrentUser_DB.P_Camera AT %DB11.DBX71.3, 100 ms
   "CurrentUser_DB_P_CycleTime" : Bool = PLC CurrentUser_DB.P_CycleTime AT %DB11.DBX71.6, 100 ms
   "HMI_BTN_EnableCycleTime" : Bool = PLC HMI_BTN_EnableCycleTime AT %M56.4, 100 ms
   "CycleTime_DB_EnabledMeasuring" : Bool = PLC CycleTime_DB.EnabledMeasuring, 100 ms
   "CycleTime_DB_CurrentPieceCognexID" : Int = PLC CycleTime_DB.CurrentPieceCognexID, 100 ms
   "CycleTime_DB_ElapsedTime_s" : Time = PLC CycleTime_DB.ElapsedTime_s, 100 ms
   "CycleTime_DB_TargetTimeInput_ms" : UInt = PLC CycleTime_DB.TargetTimeInput_ms, 1 s
   "HMI_BTN_CycleTime" : Bool = PLC HMI_BTN_CycleTime AT %M56.3, 1 s

text list "Flavors": 0 'Chocolate'; 1 'Vainilla'; 2 'Strawberry'; -1 'Flavor'; -1 'NA'

Template "Template_1" 800x480
   TextField "Template_Text field_1" at 62,8 size 412x56; Text 'MR2007B Automation of Manufacturing Systems ATOLE S.A. de C.V.'
   GraphicView "Template_Graphic view_1" at 529,9 size 252x54; Picture "eic"
   GraphicView "Template_Graphic view_2" at 21,13 size 34x45; Picture "atoleLogo_transparent"

screen "Root screen" 800x480, template "Template_1"
   TextField "HmiScreenItemData" at 40,64 size 720x57; Text 'Welcome to ATOLE S.A. de C.V.'
   GraphicView "Graphic view_1" at 400,128 size 294x294; Picture "strawberryCake"
   Button "Button_2" at 160,128 size 240x56; TextOff 'Plant View'
      on Press: SetBit("HMI_BTN_PlantView")
      on Release: ResetBit("HMI_BTN_PlantView")
   Button "Button_3" at 160,192 size 240x56; TextOff 'Set Process Times'
      on Press: SetBit("HMI_BTN_ProcessTimes")
      on Release: ResetBit("HMI_BTN_ProcessTimes")
   Button "Button_4" at 160,256 size 240x56; TextOff 'Manual Control'
      on Press: SetBit("HMI_BTN_ManualModeScr")
      on Release: ResetBit("HMI_BTN_ManualModeScr")
   Button "Button_1" at 161,321 size 240x56; TextOff 'Camera'
      on Press: SetBit("HMI_BTN_CameraControl")
      on Release: ResetBit("HMI_BTN_CameraControl")
   Button "Button_5" at 16,424 size 112x40; TextOff 'Logout'
      on Press: SetBit("HMI_BTN_Logout")
      on Release: ResetBit("HMI_BTN_Logout")
   Rectangle "Rectangle_1" at 168,136 size 40x40
      Appearance <- "CurrentUser_DB_P_PlantView"
   Rectangle "Rectangle_2" at 168,200 size 40x40
      Appearance <- "CurrentUser_DB_P_ProcessTimes"
   Rectangle "Rectangle_3" at 168,264 size 40x40
      Appearance <- "CurrentUser_DB_P_ManualControl"
   Rectangle "Rectangle_4" at 168,328 size 40x40
      Appearance <- "CurrentUser_DB_P_Camera"
   Button "Button_6" at 160,384 size 240x56; TextOff 'Get Cycle Time'
      on Press: SetBit("HMI_BTN_CycleTime")
      on Release: ResetBit("HMI_BTN_CycleTime")
   Rectangle "Rectangle_5" at 168,392 size 40x40
      Appearance <- "CurrentUser_DB_P_CycleTime"

screen "Pneumatic_Monitoring" 800x480, template "Template_1"
   GraphicView "Graphic view_1" at 76,81 size 593x386; Picture "pneumaticCellDiagram"
   Circle "Circle_8" at 384,112 size 17x17
      Visibility <- "Vertical_Piston"
   Circle "Circle_1" at 621,175 size 17x17
      Visibility <- "Conveyor1"
   Circle "Circle_2" at 80,274 size 17x17
      Visibility <- "Cntrcn_Piston_Start"
   Circle "Circle_3" at 137,273 size 17x17
      Visibility <- "Ext_Piston_Start"
   Circle "Circle_4" at 452,370 size 17x17
      Visibility <- "Turntable"
   Circle "Circle_5" at 599,270 size 17x17
      Visibility <- "Ext_Piston_Conveyor"
   Circle "Circle_6" at 632,270 size 17x17
      Visibility <- "Cntrcn_Piston_Conveyor"
   IOField "I/O field_1" at 92,91 size 138x51; FormatPattern 99.99; Unit  psi
      ProcessValue <- "pressureValue"
   IOField "I/O field_2" at 600,432 size 184x32; FormatPattern 999999999999; Unit  W
      ProcessValue <- "Power_consumption"
   TextField "Text field_2" at 616,408 size 168x23; Text 'Power Consumption'
   Button "Button_1" at 16,424 size 104x40; TextOff 'Home'
      on Press: ActivateScreen("Root screen", 0); SetTag("HMI_SetScreen", 2)
   TextField "Text field_1" at 319,67 size 162x39; Text 'Plant View'

screen "Manual_Control" 800x480, template "Template_1"
   TextField "Text field_1" at 204,95 size 393x39; Text 'Pneumatic Manual Control'
   Button "Button_1" at 16,424 size 104x40; TextOff 'Home'
      on Press: ActivateScreen("Root screen", 0); SetTag("HMI_SetScreen", 2)
   TextField "Text field_3" at 200,96 size 16x23; Text 'Text'
   TextField "Text field_2" at 56,304 size 137x36; Text 'Enable manual control'
   Button "Button_2" at 232,192 size 192x32; TextOff 'Ex. Piston Start'
      on Press: SetBit("HMI_BTN_Ext_Piston_Start")
      on Release: ResetBit("HMI_BTN_Ext_Piston_Start")
   Button "Button_3" at 232,240 size 192x32; TextOff 'C. Piston Start'
      on Press: SetBit("HMI_BTN_Cntrcn_Piston_Start")
      on Release: ResetBit("HMI_BTN_Cntrcn_Piston_Start")
   Button "Button_4" at 232,288 size 192x32; TextOff 'Vertical Piston'
      on Press: SetBit("HMI_BTN_Vertical_Piston")
      on Release: ResetBit("HMI_BTN_Vertical_Piston")
   Button "Button_5" at 232,336 size 192x32; TextOff 'Turntable'
      on Press: SetBit("HMI_BTN_Turntable")
      on Release: ResetBit("HMI_BTN_Turntable")
   Button "Button_6" at 504,192 size 192x32; TextOff 'Ex. Piston Conveyor'
      on Press: SetBit("HMI_BTN_Ext_Piston_Conveyor")
      on Release: ResetBit("HMI_BTN_Ext_Piston_Conveyor")
   Button "Button_7" at 504,240 size 192x32; TextOff 'C. Piston Conveyor'
      on Press: SetBit("HMI_BTN_Cntrcn_Piston_Conveyor")
      on Release: ResetBit("HMI_BTN_Cntrcn_Piston_Conveyor")
   Button "Button_8" at 504,288 size 192x32; TextOff 'Conveyor 1'
      on Press: SetBit("HMI_BTN_Conveyor1")
      on Release: ResetBit("HMI_BTN_Conveyor1")
   Circle "Circle_1" at 440,192 size 32x32
      Appearance <- "Ext_Piston_Start"
   Circle "Circle_2" at 440,240 size 32x32
      Appearance <- "Cntrcn_Piston_Start"
   Circle "Circle_3" at 440,288 size 32x32
      Appearance <- "Vertical_Piston"
   Circle "Circle_4" at 440,336 size 32x32
      Appearance <- "Turntable"
   Circle "Circle_5" at 712,192 size 32x32
      Appearance <- "Ext_Piston_Conveyor"
   Circle "Circle_6" at 712,240 size 32x32
      Appearance <- "Cntrcn_Piston_Conveyor"
   Circle "Circle_7" at 712,288 size 32x32
      Appearance <- "Conveyor1"
   Switch "Switch_1" at 56,240 size 136x56; CaptionText 'Switch'; TextOff 'OFF'; TextOn 'ON'
      on SwitchOn: SetBit("HMI_BTN_ManualMode")
      on SwitchOff: ResetBit("HMI_BTN_ManualMode")
   TextField "Text field_4" at 400,432 size 393x48; Text 'Manual Mode: Press and hold the button to actuate'

screen "Camera_Control" 800x480, template "Template_1"
   TextField "Text field_1" at 288,80 size 233x39; Text 'Camera Control'
   Button "Button_1" at 240,376 size 320x64; TextOff 'Scan Workpiece'
      on Press: SetBit("ScanBTN_HMI")
      on Release: ResetBit("ScanBTN_HMI")
   TextField "Text field_2" at 170,328 size 460x39; Text 'Operation in progress, wait before proceeding'
      Visibility <- "HMI_ShowBusyMessage"
   IOField "I/O field_1" at 504,136 size 168x56; FormatPattern s9
      ProcessValue <- "CognexID(1)"
   TextField "Text field_3" at 128,136 size 323x55; Text 'Scanned piece's Cognex ID'
   TextField "Text field_4" at 128,200 size 323x55; Text 'Cake flavor of scanned piece'
   SymbolicIOField "Symbolic I/O field_1" at 504,200 size 168x56; TextOff '0'; TextOn '1'; TextList "Flavors"
      ProcessValue <- "CognexID(1)"
   TextField "Text field_5" at 128,264 size 323x55; Text 'Seconds since last scan'
   IOField "I/O field_2" at 504,264 size 168x56; FormatPattern 9999999; Unit  s
      ProcessValue <- "secondsSincePhoto"
   Button "Button_3" at 16,424 size 104x40; TextOff 'Home'
      on Press: ActivateScreen("Root screen", 0); SetTag("HMI_SetScreen", 2)

screen "Process_Times" 800x480, template "Template_1"
   TextField "Text field_1" at 294,104 size 213x39; Text 'Process Times'
   Button "Button_1" at 16,424 size 104x40; TextOff 'Home'
      on Press: ActivateScreen("Root screen", 0); SetTag("HMI_SetScreen", 2)
   IOField "I/O field_1" at 200,240 size 152x48; FormatPattern 9999999; Unit  s
      ProcessValue <- "Pneumatic_Times_DB_chocolatePunchingInput_ms"
   IOField "I/O field_4" at 392,240 size 152x48; FormatPattern 9999999; Unit  s
      ProcessValue <- "Pneumatic_Times_DB_vanillaPunchingInput_ms"
   IOField "I/O field_5" at 584,240 size 152x48; FormatPattern 9999999; Unit  s
      ProcessValue <- "Pneumatic_Times_DB_strawberryPunchingInput_ms"
   TextField "Text field_2" at 200,200 size 156x34; Text 'Chocolate'
   TextField "Text field_3" at 392,200 size 156x34; Text 'Vanilla'
   TextField "Text field_4" at 584,200 size 152x31; Text 'Strawberry'
   TextField "Text field_6" at 64,240 size 120x48; Text 'Punching'

screen "Access_Screen" 800x480
   TextField "Text field_1" at 262,32 size 276x47; Text 'Access Control'
   TextField "Text field_2" at 96,176 size 226x71; Text 'Please present your RFID card to the reader interface'
   TextField "Text field_3" at 392,136 size 226x29; Text 'Current User:'
   GraphicView "Graphic view_1" at 128,232 size 160x152; Picture "rfidSym"
   Button "Button_1" at 448,328 size 248x48; TextOff 'Enter'
      on Press: SetBit("HMI_BTN_Enter")
      on Release: ResetBit("HMI_BTN_Enter")
   Circle "Circle_1" at 384,328 size 48x48
      Appearance <- "CurrentUser_DB_ValidUser"
   IOField "I/O field_1" at 384,168 size 312x48; FormatPattern ????????????????????????????????????????
      ProcessValue <- "CurrentUser_DB_Name"
   TextField "Text field_4" at 392,224 size 226x29; Text 'User role:'
   IOField "I/O field_2" at 384,256 size 312x48; FormatPattern ?????????????????????????
      ProcessValue <- "CurrentUser_DB_Role"

screen "Cycle_Time" 800x480, template "Template_1"
   Button "Button_1" at 16,424 size 104x40; TextOff 'Home'
      on Press: ActivateScreen("Root screen", 0); SetTag("HMI_SetScreen", 2)
   TextField "Text field_1" at 252,80 size 296x39; Text 'Measure Cycle Time'
   Button "Button_2" at 136,152 size 304x56; TextOff 'Enable Measuring'
      on Press: SetBit("HMI_BTN_EnableCycleTime")
      on Release: ResetBit("HMI_BTN_EnableCycleTime")
   Circle "Circle_1" at 392,160 size 40x40
      Appearance <- "CycleTime_DB_EnabledMeasuring"
   IOField "I/O field_1" at 136,224 size 304x56; FormatPattern 9999999; Unit  s
      ProcessValue <- "CycleTime_DB_ElapsedTime_s"
   TextField "Text field_2" at 144,236 size 151x29; Text 'Elapsed Time:'
   IOField "I/O field_2" at 136,296 size 304x56; FormatPattern s9
      ProcessValue <- "CycleTime_DB_CurrentPieceCognexID"
   TextField "Text field_3" at 152,309 size 100x29; Text 'Piece ID:'
   TextField "Text field_4" at 136,381 size 179x29; Text 'Set Target Time:'
   IOField "I/O field_3" at 328,368 size 112x56; FormatPattern 999999; Unit  s
      ProcessValue <- "CycleTime_DB_TargetTimeInput_ms"
   TextField "Text field_5" at 468,163 size 183x244; Text 'Instructions: 1. Confirm no pieces are currently in process. 2. Press Enable to activate cycle time measurement. 3. Go to the Camera Screen and scan a workpiece to start a sequence. 4. Wait for the sequence to finish completely before scanning the next piece.'
*)